TYPE E_MachineMode :
(
	MACHINEMODE_UNDEFINED := 0,
	MACHINEMODE_Config,
	MACHINEMODE_Init,
	MACHINEMODE_Manu,
	MACHINEMODE_SemiAuto,
	MACHINEMODE_Auto,
	MACHINEMODE_Maintenance
)USINT;
END_TYPE

(* stored: Version 1.1.0.1, ProductVersion 3.1.0.25
   DUT E_MachineMode: Id {df616623-9504-414d-a906-aef6f91d26e5} *)
